SUBAPPLICATION AUI_AX_SEL_AUI_fix (* binary selection *)
  (* Standard: 61499-2; Description: Copyright (c) 2026 HR Agrartechnik GmbH This program and the accompanying materials are made available under the terms of the Eclipse Public License 2.0 which is available at https://www.eclipse.org/legal/epl-2.0/ SPDX-License-Identifier: EPL-2.0 *)
  (* Version 1.0, 2026-04-19, Franz Höpfinger, HR Agrartechnik GmbH, initial API and implementation *)
  PACKAGE MyLib::fix;
  IMPORT eclipse4diac::core::TypeHash;
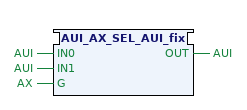
  SOCKETS
    IN0 : adapter::types::unidirectional::AUI; (* Selectable input variable *)
    IN1 : adapter::types::unidirectional::AUI; (* Selectable input variable *)
    G : adapter::types::unidirectional::AX; (* Selector *)
  END_SOCKETS
  PLUGS
    OUT : adapter::types::unidirectional::AUI; (* Selected Output *)
  END_PLUGS
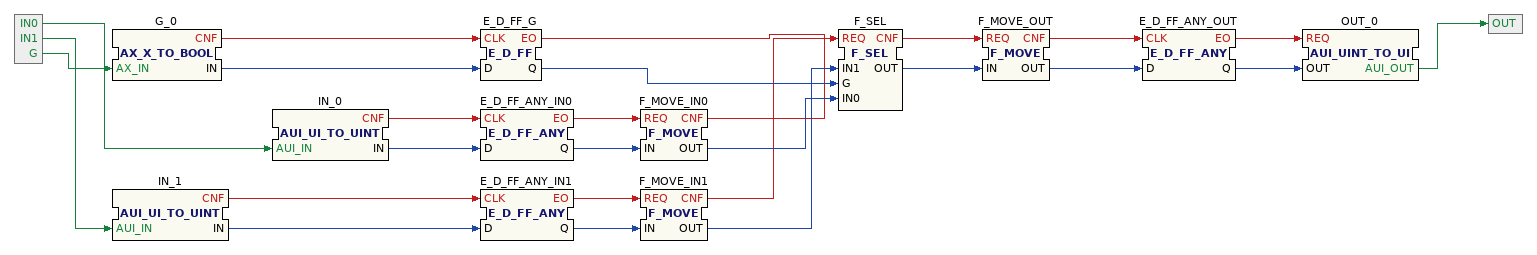
  FBS
    IN_0 : adapter::conversion::unidirectional::AUI_UI_TO_UINT;
    OUT_0 : adapter::conversion::unidirectional::AUI_UINT_TO_UI;
    IN_1 : adapter::conversion::unidirectional::AUI_UI_TO_UINT;
    G_0 : adapter::conversion::unidirectional::AX_X_TO_BOOL;
    E_D_FF_ANY_IN0 : iec61499::events::E_D_FF_ANY;
    F_MOVE_IN1 : iec61131::selection::F_MOVE; {SET_ATTRIBUTE(DataType, UINT)}
    E_D_FF_G : iec61499::events::E_D_FF;
    F_MOVE_IN0 : iec61131::selection::F_MOVE; {SET_ATTRIBUTE(DataType, UINT)}
    F_SEL : iec61131::selection::F_SEL;
    F_MOVE_OUT : iec61131::selection::F_MOVE; {SET_ATTRIBUTE(DataType, UINT)}
    E_D_FF_ANY_OUT : iec61499::events::E_D_FF_ANY;
    E_D_FF_ANY_IN1 : iec61499::events::E_D_FF_ANY;
  END_FBS
  EVENT_CONNECTIONS
    F_MOVE_IN1.CNF TO F_SEL.REQ;
    F_MOVE_OUT.CNF TO E_D_FF_ANY_OUT.CLK;
    E_D_FF_ANY_IN0.EO TO F_MOVE_IN0.REQ;
    F_SEL.CNF TO F_MOVE_OUT.REQ;
    E_D_FF_ANY_IN1.EO TO F_MOVE_IN1.REQ;
    E_D_FF_G.EO TO F_SEL.REQ;
    F_MOVE_IN0.CNF TO F_SEL.REQ;
    E_D_FF_ANY_OUT.EO TO OUT_0.REQ;
    G_0.CNF TO E_D_FF_G.CLK;
    IN_0.CNF TO E_D_FF_ANY_IN0.CLK;
    IN_1.CNF TO E_D_FF_ANY_IN1.CLK;
  END_CONNECTIONS
  DATA_CONNECTIONS
    E_D_FF_ANY_IN1.Q TO F_MOVE_IN1.IN;
    F_MOVE_IN1.OUT TO F_SEL.IN1;
    E_D_FF_G.Q TO F_SEL.G;
    F_SEL.OUT TO F_MOVE_OUT.IN;
    F_MOVE_OUT.OUT TO E_D_FF_ANY_OUT.D;
    E_D_FF_ANY_IN0.Q TO F_MOVE_IN0.IN;
    F_MOVE_IN0.OUT TO F_SEL.IN0;
    E_D_FF_ANY_OUT.Q TO OUT_0.OUT;
    G_0.IN TO E_D_FF_G.D;
    IN_0.IN TO E_D_FF_ANY_IN0.D;
    IN_1.IN TO E_D_FF_ANY_IN1.D;
  END_CONNECTIONS
  ADAPTER_CONNECTIONS
    OUT_0.AUI_OUT TO OUT;
    G TO G_0.AX_IN;
    IN1 TO IN_1.AUI_IN;
    IN0 TO IN_0.AUI_IN;
  END_CONNECTIONS
END_SUBAPPLICATION
